VAR_GLOBAL CONSTANT
	ATM_PRESS : INT := 760; // Atmospheric pressure in Torr
	ATM_PRESS_ERR_RNG : INT := 10; // Error range that is still considered atmospheric pressure
	
	EPICS_STRING_SIZE : INT := 40;
	PTM_INTERLOCK_SP : REAL := 1E-2;
END_VAR

(* stored: Version 1.1.0.1, ProductVersion 3.1.4022.18
   GVL GVL_Constants: Id {d11ce1ce-67df-4050-b028-330096f17141} *)
